Staubli VAL3: stringtopoint.pgx

program stringtopoint(string x_sString, num x_nNum)
  local bool l_btest
  local num l_nNum6
  local string l_s
  local num nA
  local num nB
  local num nC
  local num nX
  local num nY
  local num nZ
  local pointRx pChangeMid1
  local pointRx pChangeMid2
  local trsf tTrsf
begin
  l_s=x_sString
  l_s=toNum(l_s,nX,l_btest)
  l_s=toNum(l_s,nY,l_btest)
  l_s=toNum(l_s,nZ,l_btest)
  l_s=toNum(l_s,nA,l_btest)
  l_s=toNum(l_s,nB,l_btest)
  l_s=toNum(l_s,nC,l_btest)
  pfrmCad[x_nNum].trsf={nX,nY,nZ,nA,nB,nC}
  link(pfrmCad[x_nNum],FrmDraw)
end
